// TIA Portal V18 export
// export: Created 2026-06-12T02:00:00Z, ExportSetting WithDefaults, DisplayName Totally Integrated Automation Portal, DisplayVersion V18, DisplayName TIA Portal Openness, DisplayVersion V18
TagTable "HMI_Tags_B3to7"
  AI_B3_Sequence_Count : Real  (PLC tag AI_B3_Sequence_Count, HMI_Connection_1, 1 s)   // 0-100
  AI_B3_Flow_CIP_Center : Real  (PLC tag AI_B3_Flow_CIP_Center, HMI_Connection_1, 1 s)   // 100-200 L/h
  AI_B3_Temp_CIP_Upper : Real  (PLC tag AI_B3_Temp_CIP_Upper, HMI_Connection_1, 1 s)   // 50-80 °C
  AI_B3_Pressure_CIP_1 : Real  (PLC tag AI_B3_Pressure_CIP_1, HMI_Connection_1, 1 s)   // 7.0-8.0 bar
  AI_B3_Temp_Chaff_1 : Real  (PLC tag AI_B3_Temp_Chaff_1, HMI_Connection_1, 1 s)   // 50-80 °C
  AI_B3_Flow_CIP_Feed : Real  (PLC tag AI_B3_Flow_CIP_Feed, HMI_Connection_1, 1 s)   // 100-200 L/h
  AI_B3_Temp_Steam_1 : Real  (PLC tag AI_B3_Temp_Steam_1, HMI_Connection_1, 1 s)   // 50-80 °C
  AI_B3_Flow_UCWW_1 : Real  (PLC tag AI_B3_Flow_UCWW_1, HMI_Connection_1, 1 s)   // 100-200 L/h
  AI_B3_RPM_Screw_Conv : Real  (PLC tag AI_B3_RPM_Screw_Conv, HMI_Connection_1, 1 s)   // 800-1200 RPM
  AI_B3_Temp_Condensate_1 : Real  (PLC tag AI_B3_Temp_Condensate_1, HMI_Connection_1, 1 s)   // 50-80 °C
  AI_B3_Pressure_Screw_1 : Real  (PLC tag AI_B3_Pressure_Screw_1, HMI_Connection_1, 1 s)   // 7.0-8.0 bar
  AI_B3_Flow_CWW_Out : Real  (PLC tag AI_B3_Flow_CWW_Out, HMI_Connection_1, 1 s)   // 100-200 L/h
  AI_B3_Pressure_CWW_1 : Real  (PLC tag AI_B3_Pressure_CWW_1, HMI_Connection_1, 1 s)   // 7.0-8.0 bar
  AI_B3_Temp_Decanter2 : Real  (PLC tag AI_B3_Temp_Decanter2, HMI_Connection_1, 1 s)   // 50-80 °C
  AI_B3_RPM_Rotary2 : Real  (PLC tag AI_B3_RPM_Rotary2, HMI_Connection_1, 1 s)   // 800-1200 RPM
  AI_B3_RPM_Rotary1 : Real  (PLC tag AI_B3_RPM_Rotary1, HMI_Connection_1, 1 s)   // 800-1200 RPM
  AI_B3_Temp_GroundSilo : Real  (PLC tag AI_B3_Temp_GroundSilo, HMI_Connection_1, 1 s)   // 50-80 °C
  AI_B3_Flow_GroundSilo : Real  (PLC tag AI_B3_Flow_GroundSilo, HMI_Connection_1, 1 s)   // 100-200 L/h
  AI_B3_Pressure_Mid_1 : Real  (PLC tag AI_B3_Pressure_Mid_1, HMI_Connection_1, 1 s)   // 7.0-8.0 bar
  AI_B3_Flow_Condensate : Real  (PLC tag AI_B3_Flow_Condensate, HMI_Connection_1, 1 s)   // 100-200 L/h
  AI_B3_Flow_Sump_Out : Real  (PLC tag AI_B3_Flow_Sump_Out, HMI_Connection_1, 1 s)   // 100-200 L/h
  AI_B3_Level_Sump : Real  (PLC tag AI_B3_Level_Sump, HMI_Connection_1, 1 s)   // 30-80 %
  AI_B3_Pressure_Decant1 : Real  (PLC tag AI_B3_Pressure_Decant1, HMI_Connection_1, 1 s)   // 7.0-8.0 bar
  AI_B3_Pressure_Decant2 : Real  (PLC tag AI_B3_Pressure_Decant2, HMI_Connection_1, 1 s)   // 7.0-8.0 bar
  AI_B3_Flow_Decant1 : Real  (PLC tag AI_B3_Flow_Decant1, HMI_Connection_1, 1 s)   // 100-200 L/h
  AI_B3_Temp_Decant1 : Real  (PLC tag AI_B3_Temp_Decant1, HMI_Connection_1, 1 s)   // 50-80 °C
  AI_B3_Temp_FBB_Boiler : Real  (PLC tag AI_B3_Temp_FBB_Boiler, HMI_Connection_1, 1 s)   // 50-80 °C
  AI_B3_Temp_CWW_Out : Real  (PLC tag AI_B3_Temp_CWW_Out, HMI_Connection_1, 1 s)   // 50-80 °C
  AI_B3_Pressure_SUMP : Real  (PLC tag AI_B3_Pressure_SUMP, HMI_Connection_1, 1 s)   // 7.0-8.0 bar
  AI_B3_Flow_SUMP : Real  (PLC tag AI_B3_Flow_SUMP, HMI_Connection_1, 1 s)   // 100-200 L/h
  AI_B3_Level_CWW : Real  (PLC tag AI_B3_Level_CWW, HMI_Connection_1, 1 s)   // 30-80 %
  AI_B3_Temp_FBB_Out : Real  (PLC tag AI_B3_Temp_FBB_Out, HMI_Connection_1, 1 s)   // 50-80 °C
  AI_B3_Pressure_FBB_Out : Real  (PLC tag AI_B3_Pressure_FBB_Out, HMI_Connection_1, 1 s)   // 7.0-8.0 bar
  AI_B3_Flow_FBB_Out : Real  (PLC tag AI_B3_Flow_FBB_Out, HMI_Connection_1, 1 s)   // 100-200 L/h
  AI_B4_Daq_C : Real  (PLC tag AI_B4_Daq_C, HMI_Connection_1, 1 s)   // 0-100
  AI_B4_TPH_Total : Real  (PLC tag AI_B4_TPH_Total, HMI_Connection_1, 1 s)   // 100-200 T/h
  AI_B4_KG_CM_Main : Real  (PLC tag AI_B4_KG_CM_Main, HMI_Connection_1, 1 s)   // 7.0-8.0 kg/cm2
  AI_B4_DRM_LVL1 : Real  (PLC tag AI_B4_DRM_LVL1, HMI_Connection_1, 1 s)   // 30-80 %
  AI_B4_DRM_LVL2 : Real  (PLC tag AI_B4_DRM_LVL2, HMI_Connection_1, 1 s)   // 30-80 %
  AI_B4_MW_Output : Real  (PLC tag AI_B4_MW_Output, HMI_Connection_1, 1 s)   // 0-50 MW
  AI_B4_KG_CM_2 : Real  (PLC tag AI_B4_KG_CM_2, HMI_Connection_1, 1 s)   // 7.0-8.0 kg/cm2
  AI_B4_Hc_Value : Real  (PLC tag AI_B4_Hc_Value, HMI_Connection_1, 1 s)   // 0-100
  AI_B4_Temp_AirHeater_In1 : Real  (PLC tag AI_B4_Temp_AirHeater_In1, HMI_Connection_1, 1 s)   // 50-80 °C
  AI_B4_Temp_AirHeater_In2 : Real  (PLC tag AI_B4_Temp_AirHeater_In2, HMI_Connection_1, 1 s)   // 50-80 °C
  AI_B4_Temp_AirHeater_In3 : Real  (PLC tag AI_B4_Temp_AirHeater_In3, HMI_Connection_1, 1 s)   // 50-80 °C
  AI_B4_Temp_AirHeater_Out1 : Real  (PLC tag AI_B4_Temp_AirHeater_Out1, HMI_Connection_1, 1 s)   // 50-80 °C
  AI_B4_Temp_AirHeater_Out2 : Real  (PLC tag AI_B4_Temp_AirHeater_Out2, HMI_Connection_1, 1 s)   // 50-80 °C
  AI_B4_Pres_AH_mmWC_1 : Real  (PLC tag AI_B4_Pres_AH_mmWC_1, HMI_Connection_1, 1 s)   // 7.0-8.0 mmWC
  AI_B4_Pres_AH_mmWC_2 : Real  (PLC tag AI_B4_Pres_AH_mmWC_2, HMI_Connection_1, 1 s)   // 7.0-8.0 mmWC
  AI_B4_Pres_AH_Pct_1 : Real  (PLC tag AI_B4_Pres_AH_Pct_1, HMI_Connection_1, 1 s)   // 20-80 %
  AI_B4_Temp_AH_Out3 : Real  (PLC tag AI_B4_Temp_AH_Out3, HMI_Connection_1, 1 s)   // 50-80 °C
  AI_B4_Pres_FDH_mmWC : Real  (PLC tag AI_B4_Pres_FDH_mmWC, HMI_Connection_1, 1 s)   // 7.0-8.0 mmWC
  AI_B4_RPM_PAF1 : Real  (PLC tag AI_B4_RPM_PAF1, HMI_Connection_1, 1 s)   // 800-1200 RPM
  AI_B4_Pct_RPC308_SP : Real  (PLC tag AI_B4_Pct_RPC308_SP, HMI_Connection_1, 1 s)   // 20-80 %
  AI_B4_Pct_RPC308_PV : Real  (PLC tag AI_B4_Pct_RPC308_PV, HMI_Connection_1, 1 s)   // 20-80 %
  AI_B4_Pres_PAF1_mmWC : Real  (PLC tag AI_B4_Pres_PAF1_mmWC, HMI_Connection_1, 1 s)   // 7.0-8.0 mmWC
  AI_B4_Pct_FDF1_SP : Real  (PLC tag AI_B4_Pct_FDF1_SP, HMI_Connection_1, 1 s)   // 20-80 %
  AI_B4_Pct_FDF1_PV : Real  (PLC tag AI_B4_Pct_FDF1_PV, HMI_Connection_1, 1 s)   // 20-80 %
  AI_B4_Pct_FDF1_OUT : Real  (PLC tag AI_B4_Pct_FDF1_OUT, HMI_Connection_1, 1 s)   // 20-80 %
  AI_B4_RPM_FDF1 : Real  (PLC tag AI_B4_RPM_FDF1, HMI_Connection_1, 1 s)   // 800-1200 RPM
  AI_B4_Pct_RPC301_SP : Real  (PLC tag AI_B4_Pct_RPC301_SP, HMI_Connection_1, 1 s)   // 20-80 %
  AI_B4_Pct_RPC301_PV : Real  (PLC tag AI_B4_Pct_RPC301_PV, HMI_Connection_1, 1 s)   // 20-80 %
  AI_B4_Pct_RPC301_OUT : Real  (PLC tag AI_B4_Pct_RPC301_OUT, HMI_Connection_1, 1 s)   // 20-80 %
  AI_B4_mA_ESP1 : Real  (PLC tag AI_B4_mA_ESP1, HMI_Connection_1, 1 s)   // 50-200 mA
  AI_B4_mA_ESP2 : Real  (PLC tag AI_B4_mA_ESP2, HMI_Connection_1, 1 s)   // 50-200 mA
  AI_B4_mA_ESP3 : Real  (PLC tag AI_B4_mA_ESP3, HMI_Connection_1, 1 s)   // 50-200 mA
  AI_B4_mA_ESP4 : Real  (PLC tag AI_B4_mA_ESP4, HMI_Connection_1, 1 s)   // 50-200 mA
  AI_B4_V_ESP1 : Real  (PLC tag AI_B4_V_ESP1, HMI_Connection_1, 1 s)   // 0-400 V
  AI_B4_V_ESP2 : Real  (PLC tag AI_B4_V_ESP2, HMI_Connection_1, 1 s)   // 0-400 V
  AI_B4_V_ESP3 : Real  (PLC tag AI_B4_V_ESP3, HMI_Connection_1, 1 s)   // 0-400 V
  AI_B4_V_ESP4 : Real  (PLC tag AI_B4_V_ESP4, HMI_Connection_1, 1 s)   // 0-400 V
  AI_B4_Pct_RPC305_SP : Real  (PLC tag AI_B4_Pct_RPC305_SP, HMI_Connection_1, 1 s)   // 20-80 %
  AI_B4_Pct_RPC305_PV : Real  (PLC tag AI_B4_Pct_RPC305_PV, HMI_Connection_1, 1 s)   // 20-80 %
  AI_B4_RPM_IDF1 : Real  (PLC tag AI_B4_RPM_IDF1, HMI_Connection_1, 1 s)   // 800-1200 RPM
  AI_B4_Pct_RPC305_VFD : Real  (PLC tag AI_B4_Pct_RPC305_VFD, HMI_Connection_1, 1 s)   // 20-80 %
  AI_B4_Pct_FDF2_SP : Real  (PLC tag AI_B4_Pct_FDF2_SP, HMI_Connection_1, 1 s)   // 20-80 %
  AI_B4_Pct_FDF2_PV : Real  (PLC tag AI_B4_Pct_FDF2_PV, HMI_Connection_1, 1 s)   // 20-80 %
  AI_B4_Pct_FDF2_OUT : Real  (PLC tag AI_B4_Pct_FDF2_OUT, HMI_Connection_1, 1 s)   // 20-80 %
  AI_B4_RPM_FDF2 : Real  (PLC tag AI_B4_RPM_FDF2, HMI_Connection_1, 1 s)   // 800-1200 RPM
  AI_B4_Pct_RPC306_SP : Real  (PLC tag AI_B4_Pct_RPC306_SP, HMI_Connection_1, 1 s)   // 20-80 %
  AI_B4_Pct_RPC306_PV : Real  (PLC tag AI_B4_Pct_RPC306_PV, HMI_Connection_1, 1 s)   // 20-80 %
  AI_B4_Pct_RPC306_OUT : Real  (PLC tag AI_B4_Pct_RPC306_OUT, HMI_Connection_1, 1 s)   // 20-80 %
  AI_B4_RPM_IDF2 : Real  (PLC tag AI_B4_RPM_IDF2, HMI_Connection_1, 1 s)   // 800-1200 RPM
  AI_B4_Pct_RPC306_VFD : Real  (PLC tag AI_B4_Pct_RPC306_VFD, HMI_Connection_1, 1 s)   // 20-80 %
  AI_B4_Pres_FDF_mmWC : Real  (PLC tag AI_B4_Pres_FDF_mmWC, HMI_Connection_1, 1 s)   // 7.0-8.0 mmWC
  AI_B4_TEST1_Value : Real  (PLC tag AI_B4_TEST1_Value, HMI_Connection_1, 1 s)   // 0-100
  AI_B4_Pct_PAF1_SP : Real  (PLC tag AI_B4_Pct_PAF1_SP, HMI_Connection_1, 1 s)   // 20-80 %
  AI_B4_Pct_PAF1_PV : Real  (PLC tag AI_B4_Pct_PAF1_PV, HMI_Connection_1, 1 s)   // 20-80 %
  AI_B4_Pres_PAF2_mmWC : Real  (PLC tag AI_B4_Pres_PAF2_mmWC, HMI_Connection_1, 1 s)   // 7.0-8.0 mmWC
  AI_B4_RPM_PAF2 : Real  (PLC tag AI_B4_RPM_PAF2, HMI_Connection_1, 1 s)   // 800-1200 RPM
  AI_B4_Pct_RPC308b_SP : Real  (PLC tag AI_B4_Pct_RPC308b_SP, HMI_Connection_1, 1 s)   // 20-80 %
  AI_B4_Pct_RPC308b_PV : Real  (PLC tag AI_B4_Pct_RPC308b_PV, HMI_Connection_1, 1 s)   // 20-80 %
  AI_B4_Pct_DAM303B_SP : Real  (PLC tag AI_B4_Pct_DAM303B_SP, HMI_Connection_1, 1 s)   // 20-80 %
  AI_B4_Pct_DAM304B_SP : Real  (PLC tag AI_B4_Pct_DAM304B_SP, HMI_Connection_1, 1 s)   // 20-80 %
  AI_B5_CA_Fan_Motor_DE_Temp : Real  (PLC tag AI_B5_CA_Fan_Motor_DE_Temp, HMI_Connection_1, 1 s)   // 50-80 °C
  AI_B5_CA_Fan_Motor_NDE_Temp : Real  (PLC tag AI_B5_CA_Fan_Motor_NDE_Temp, HMI_Connection_1, 1 s)   // 50-80 °C
  AI_B5_CA_Fan_DE_Temp : Real  (PLC tag AI_B5_CA_Fan_DE_Temp, HMI_Connection_1, 1 s)   // 50-80 °C
  AI_B5_CA_Fan_NDE_Temp : Real  (PLC tag AI_B5_CA_Fan_NDE_Temp, HMI_Connection_1, 1 s)   // 50-80 °C
  AI_B5_CA_Fan_DE_Vib : Real  (PLC tag AI_B5_CA_Fan_DE_Vib, HMI_Connection_1, 1 s)   // 0-10 mm/s
  AI_B5_CA_Fan_NDE_Vib : Real  (PLC tag AI_B5_CA_Fan_NDE_Vib, HMI_Connection_1, 1 s)   // 0-10 mm/s
  AI_B5_SP_700FN03 : Real  (PLC tag AI_B5_SP_700FN03, HMI_Connection_1, 1 s)   // 100-200 L/h
  AI_B5_SP_700HES01 : Real  (PLC tag AI_B5_SP_700HES01, HMI_Connection_1, 1 s)   // 100-200 L/h
  AI_B5_SP_700DA4 : Real  (PLC tag AI_B5_SP_700DA4, HMI_Connection_1, 1 s)   // 20-30 Hz
  AI_B5_SP_700DA6 : Real  (PLC tag AI_B5_SP_700DA6, HMI_Connection_1, 1 s)   // 20-30 Hz
  AI_B5_SP_700DA7 : Real  (PLC tag AI_B5_SP_700DA7, HMI_Connection_1, 1 s)   // 20-30 Hz
  AI_B5_SP_700FN2_DA1 : Real  (PLC tag AI_B5_SP_700FN2_DA1, HMI_Connection_1, 1 s)   // 20-30 Hz
  AI_B5_Sep_Motor_Top_Temp : Real  (PLC tag AI_B5_Sep_Motor_Top_Temp, HMI_Connection_1, 1 s)   // 50-80 °C
  AI_B5_Sep_Bottom_Bear_Temp : Real  (PLC tag AI_B5_Sep_Bottom_Bear_Temp, HMI_Connection_1, 1 s)   // 50-80 °C
  AI_B5_Trend_Val_1 : Real  (PLC tag AI_B5_Trend_Val_1, HMI_Connection_1, 1 s)   // 0-100 %
  AI_B5_Trend_Val_2 : Real  (PLC tag AI_B5_Trend_Val_2, HMI_Connection_1, 1 s)   // 0-100 %
  AI_B5_Trend_Val_3 : Real  (PLC tag AI_B5_Trend_Val_3, HMI_Connection_1, 1 s)   // 0-100 %
  AI_B5_700FN03_RPM : Real  (PLC tag AI_B5_700FN03_RPM, HMI_Connection_1, 1 s)   // 800-1200 RPM
  AI_B5_700HES01_Flow : Real  (PLC tag AI_B5_700HES01_Flow, HMI_Connection_1, 1 s)   // 100-200 L/h
  AI_B5_700FN10_Speed : Real  (PLC tag AI_B5_700FN10_Speed, HMI_Connection_1, 1 s)   // 20-30 Hz
  AI_B5_700CM01_Current : Real  (PLC tag AI_B5_700CM01_Current, HMI_Connection_1, 1 s)   // 50-200 A
  AI_B5_Lub_Stop_Time : Real  (PLC tag AI_B5_Lub_Stop_Time, HMI_Connection_1, 1 s)   // 0-300 Sec
  AI_B5_Main_Drive_ReHealth : Real  (PLC tag AI_B5_Main_Drive_ReHealth, HMI_Connection_1, 1 s)   // 0-300 Sec
  AI_B5_CM_LRS_IN : Real  (PLC tag AI_B5_CM_LRS_IN, HMI_Connection_1, 1 s)   // 50-80 °C
  AI_B5_CM_LRS_OUT : Real  (PLC tag AI_B5_CM_LRS_OUT, HMI_Connection_1, 1 s)   // 50-80 °C
  AI_B5_CM_Mill_Oil_Temp : Real  (PLC tag AI_B5_CM_Mill_Oil_Temp, HMI_Connection_1, 1 s)   // 50-80 °C
  AI_B5_CM_OilTrun_BER_Temp : Real  (PLC tag AI_B5_CM_OilTrun_BER_Temp, HMI_Connection_1, 1 s)   // 50-80 °C
  AI_B5_CM_OilTrun_BER2_Temp : Real  (PLC tag AI_B5_CM_OilTrun_BER2_Temp, HMI_Connection_1, 1 s)   // 50-80 °C
  AI_B5_CM_OilPinion_BER_Temp : Real  (PLC tag AI_B5_CM_OilPinion_BER_Temp, HMI_Connection_1, 1 s)   // 50-80 °C
  AI_B5_CM_GB_IL_Shaft_BER : Real  (PLC tag AI_B5_CM_GB_IL_Shaft_BER, HMI_Connection_1, 1 s)   // 50-80 °C
  AI_B5_CM_Running_Hours : Real  (PLC tag AI_B5_CM_Running_Hours, HMI_Connection_1, 1 s)   // 0-8760 Hr
  AI_B5_CM_PS1_1_KG : Real  (PLC tag AI_B5_CM_PS1_1_KG, HMI_Connection_1, 1 s)   // 7-8 bar
  AI_B5_CM_PS1_2_KG : Real  (PLC tag AI_B5_CM_PS1_2_KG, HMI_Connection_1, 1 s)   // 7-8 bar
  AI_B5_NIBS_Value : Real  (PLC tag AI_B5_NIBS_Value, HMI_Connection_1, 1 s)   // 50-200 A
  AI_B5_800DC1_Temp : Real  (PLC tag AI_B5_800DC1_Temp, HMI_Connection_1, 1 s)   // 50-80 °C
  AI_B5_800DC2_Temp : Real  (PLC tag AI_B5_800DC2_Temp, HMI_Connection_1, 1 s)   // 50-80 °C
  AI_B5_800FN1_Speed : Real  (PLC tag AI_B5_800FN1_Speed, HMI_Connection_1, 1 s)   // 20-30 Hz
  AI_B5_800FN2_Speed : Real  (PLC tag AI_B5_800FN2_Speed, HMI_Connection_1, 1 s)   // 20-30 Hz
  AI_B5_800YF1_Flow : Real  (PLC tag AI_B5_800YF1_Flow, HMI_Connection_1, 1 s)   // 100-200 L/h
  AI_B5_800YF2_Flow : Real  (PLC tag AI_B5_800YF2_Flow, HMI_Connection_1, 1 s)   // 100-200 L/h
  AI_B5_Silo1_Level_Bar1 : Real  (PLC tag AI_B5_Silo1_Level_Bar1, HMI_Connection_1, 1 s)   // 0-100 %
  AI_B5_Silo1_Level_Bar2 : Real  (PLC tag AI_B5_Silo1_Level_Bar2, HMI_Connection_1, 1 s)   // 0-100 %
  AI_B5_Silo2_Level_Bar1 : Real  (PLC tag AI_B5_Silo2_Level_Bar1, HMI_Connection_1, 1 s)   // 0-100 %
  AI_B5_Silo2_Level_Bar2 : Real  (PLC tag AI_B5_Silo2_Level_Bar2, HMI_Connection_1, 1 s)   // 0-100 %
  AI_B5_700FN01_Speed : Real  (PLC tag AI_B5_700FN01_Speed, HMI_Connection_1, 1 s)   // 20-30 Hz
  AI_B5_700FN02_Speed : Real  (PLC tag AI_B5_700FN02_Speed, HMI_Connection_1, 1 s)   // 20-30 Hz
  AI_B5_700AS07_Speed : Real  (PLC tag AI_B5_700AS07_Speed, HMI_Connection_1, 1 s)   // 20-30 Hz
  AI_B5_700AS08_Flow : Real  (PLC tag AI_B5_700AS08_Flow, HMI_Connection_1, 1 s)   // 100-200 L/h
  AI_B5_700FN09_Speed : Real  (PLC tag AI_B5_700FN09_Speed, HMI_Connection_1, 1 s)   // 20-30 Hz
  AI_B5_700SFM01_Speed : Real  (PLC tag AI_B5_700SFM01_Speed, HMI_Connection_1, 1 s)   // 20-30 Hz
  AI_B5_700DA1_Flow : Real  (PLC tag AI_B5_700DA1_Flow, HMI_Connection_1, 1 s)   // 100-200 L/h
  AI_B5_700DA4_Flow : Real  (PLC tag AI_B5_700DA4_Flow, HMI_Connection_1, 1 s)   // 100-200 L/h
  AI_B5_700DA6_Temp : Real  (PLC tag AI_B5_700DA6_Temp, HMI_Connection_1, 1 s)   // 50-80 °C
  AI_B5_700DA7_Temp : Real  (PLC tag AI_B5_700DA7_Temp, HMI_Connection_1, 1 s)   // 50-80 °C
  AI_B5_700BL1_Load : Real  (PLC tag AI_B5_700BL1_Load, HMI_Connection_1, 1 s)   // 50-200 A
  AI_B5_700BL2_Load : Real  (PLC tag AI_B5_700BL2_Load, HMI_Connection_1, 1 s)   // 50-200 A
  AI_B5_700AS9_Flow : Real  (PLC tag AI_B5_700AS9_Flow, HMI_Connection_1, 1 s)   // 100-200 L/h
  AI_B5_700FN13_Speed : Real  (PLC tag AI_B5_700FN13_Speed, HMI_Connection_1, 1 s)   // 20-30 Hz
  AI_B6_TICR211_Temp : Real  (PLC tag AI_B6_TICR211_Temp, HMI_Connection_1, 1 s)   // 50-80 °C
  AI_B6_TICR210_Temp : Real  (PLC tag AI_B6_TICR210_Temp, HMI_Connection_1, 1 s)   // 50-80 °C
  AI_B6_TICR201_Tank_Temp : Real  (PLC tag AI_B6_TICR201_Tank_Temp, HMI_Connection_1, 1 s)   // 50-80 °C
  AI_B6_PT201_Pressure : Real  (PLC tag AI_B6_PT201_Pressure, HMI_Connection_1, 1 s)   // 7.0-8.0 bar
  AI_B6_Ph201_pH : Real  (PLC tag AI_B6_Ph201_pH, HMI_Connection_1, 1 s)   // 6.0-8.0 pH
  AI_B6_ORP201_ORP : Real  (PLC tag AI_B6_ORP201_ORP, HMI_Connection_1, 1 s)   // 20-80 %
  AI_B6_DPL101_Level : Real  (PLC tag AI_B6_DPL101_Level, HMI_Connection_1, 1 s)   // 100-500 L
  AI_B6_TICR214_Temp : Real  (PLC tag AI_B6_TICR214_Temp, HMI_Connection_1, 1 s)   // 50-80 °C
  AI_B6_TICR204_Temp : Real  (PLC tag AI_B6_TICR204_Temp, HMI_Connection_1, 1 s)   // 50-80 °C
  AI_B6_TICR205_Temp : Real  (PLC tag AI_B6_TICR205_Temp, HMI_Connection_1, 1 s)   // 50-80 °C
  AI_B6_TICR206_Temp : Real  (PLC tag AI_B6_TICR206_Temp, HMI_Connection_1, 1 s)   // 50-80 °C
  AI_B6_FHC203_Flow : Real  (PLC tag AI_B6_FHC203_Flow, HMI_Connection_1, 1 s)   // 100-200 L/h
  AI_B6_BPC201_Pressure : Real  (PLC tag AI_B6_BPC201_Pressure, HMI_Connection_1, 1 s)   // 7.0-8.0 bar
  AI_B7_K03_PT02_Pressure : Real  (PLC tag AI_B7_K03_PT02_Pressure, HMI_Connection_1, 1 s)   // 7-8 bar
  AI_B7_K03_TT04_Temp : Real  (PLC tag AI_B7_K03_TT04_Temp, HMI_Connection_1, 1 s)   // 50-80 °C
  AI_B7_K03_TT05_Temp : Real  (PLC tag AI_B7_K03_TT05_Temp, HMI_Connection_1, 1 s)   // 50-80 °C
  AI_B7_K03_TT06_Temp : Real  (PLC tag AI_B7_K03_TT06_Temp, HMI_Connection_1, 1 s)   // 50-80 °C
  AI_B7_K03_TT07_Temp : Real  (PLC tag AI_B7_K03_TT07_Temp, HMI_Connection_1, 1 s)   // 50-80 °C
  AI_B7_K03_PT07_Pressure : Real  (PLC tag AI_B7_K03_PT07_Pressure, HMI_Connection_1, 1 s)   // 7-8 bar
  AI_B7_K03_FT03_Flow : Real  (PLC tag AI_B7_K03_FT03_Flow, HMI_Connection_1, 1 s)   // 100-200 L/h
  AI_B7_K03_Density_1 : Real  (PLC tag AI_B7_K03_Density_1, HMI_Connection_1, 1 s)   // 800-1000 kg/m3
  AI_B7_K03_LT01_Level : Real  (PLC tag AI_B7_K03_LT01_Level, HMI_Connection_1, 1 s)   // 20-80 cm
  AI_B7_K03_LT02_Level : Real  (PLC tag AI_B7_K03_LT02_Level, HMI_Connection_1, 1 s)   // 20-80 cm
  AI_B7_K03_TT01_Temp : Real  (PLC tag AI_B7_K03_TT01_Temp, HMI_Connection_1, 1 s)   // 50-80 °C
  AI_B7_K03_TT02_Temp : Real  (PLC tag AI_B7_K03_TT02_Temp, HMI_Connection_1, 1 s)   // 50-80 °C
  AI_B7_Reboiler_PV : Real  (PLC tag AI_B7_Reboiler_PV, HMI_Connection_1, 1 s)   // 100-200 L/h
  AI_B7_Reboiler_SP : Real  (PLC tag AI_B7_Reboiler_SP, HMI_Connection_1, 1 s)   // 100-200 L/h
  AI_B7_Reboiler_CV : Real  (PLC tag AI_B7_Reboiler_CV, HMI_Connection_1, 1 s)   // 20-80 %
  AI_B7_HE03_Primary_Temp : Real  (PLC tag AI_B7_HE03_Primary_Temp, HMI_Connection_1, 1 s)   // 50-80 °C
  AI_B7_HE03_Secondary_Temp : Real  (PLC tag AI_B7_HE03_Secondary_Temp, HMI_Connection_1, 1 s)   // 50-80 °C
  AI_B7_K03_L08_Level : Real  (PLC tag AI_B7_K03_L08_Level, HMI_Connection_1, 1 s)   // 20-80 cm
  AI_B7_K03_L06_Level : Real  (PLC tag AI_B7_K03_L06_Level, HMI_Connection_1, 1 s)   // 20-80 cm
  AI_B7_K03_L05_Level : Real  (PLC tag AI_B7_K03_L05_Level, HMI_Connection_1, 1 s)   // 20-80 cm
  AI_B7_K03_L07_Level : Real  (PLC tag AI_B7_K03_L07_Level, HMI_Connection_1, 1 s)   // 20-80 cm
  AI_B7_K03_L04_Level : Real  (PLC tag AI_B7_K03_L04_Level, HMI_Connection_1, 1 s)   // 20-80 cm
  AI_B7_K03_L03_Level : Real  (PLC tag AI_B7_K03_L03_Level, HMI_Connection_1, 1 s)   // 20-80 cm
  AI_B7_V03A_Density : Real  (PLC tag AI_B7_V03A_Density, HMI_Connection_1, 1 s)   // 800-1000 kg/m3
  AI_B7_Kettle_Flow_SP : Real  (PLC tag AI_B7_Kettle_Flow_SP, HMI_Connection_1, 1 s)   // 100-200 kg/h
  AI_B7_Keboiler_Flow_SP : Real  (PLC tag AI_B7_Keboiler_Flow_SP, HMI_Connection_1, 1 s)   // 100-200 kg/h
  AI_B7_Reflux_Time_SP : Real  (PLC tag AI_B7_Reflux_Time_SP, HMI_Connection_1, 1 s)   // 0-60 Min
  AI_B7_Time_Remain : Real  (PLC tag AI_B7_Time_Remain, HMI_Connection_1, 1 s)   // 0-60 Min
  AI_B7_RD_Level_SP : Real  (PLC tag AI_B7_RD_Level_SP, HMI_Connection_1, 1 s)   // 20-80 cm
  AI_B7_Reflux_Flow_SP : Real  (PLC tag AI_B7_Reflux_Flow_SP, HMI_Connection_1, 1 s)   // 100-200 L/h
  AI_B7_Collection_SP : Real  (PLC tag AI_B7_Collection_SP, HMI_Connection_1, 1 s)   // 100-200 L/h
  AI_B7_Total_Flowrate : Real  (PLC tag AI_B7_Total_Flowrate, HMI_Connection_1, 1 s)   // 100-200 L/h
  AI_B7_ML_Qty_SP : Real  (PLC tag AI_B7_ML_Qty_SP, HMI_Connection_1, 1 s)   // 0-600 L
  AI_B7_ML_Qty_Total : Real  (PLC tag AI_B7_ML_Qty_Total, HMI_Connection_1, 1 s)   // 0-600 L
  AI_B7_Material_Code : Real  (PLC tag AI_B7_Material_Code, HMI_Connection_1, 1 s)   // 0-99
  AI_B7_Stage_Number : Real  (PLC tag AI_B7_Stage_Number, HMI_Connection_1, 1 s)   // 0-20
  AI_B7_Batch_Number : Real  (PLC tag AI_B7_Batch_Number, HMI_Connection_1, 1 s)   // 0-9999
  AI_B7_Current_User_ID : Real  (PLC tag AI_B7_Current_User_ID, HMI_Connection_1, 1 s)   // 0-999
  AI_B7_K_05_L_704_HI : Real  (PLC tag AI_B7_K_05_L_704_HI, HMI_Connection_1, 1 s)   // 20-80 cm
  AI_B7_Density_SP : Real  (PLC tag AI_B7_Density_SP, HMI_Connection_1, 1 s)   // 800-1000 kg/m3
  AI_B7_CTS_Flow_1 : Real  (PLC tag AI_B7_CTS_Flow_1, HMI_Connection_1, 1 s)   // 100-200 kg/h
  AI_B7_CTS_Flow_2 : Real  (PLC tag AI_B7_CTS_Flow_2, HMI_Connection_1, 1 s)   // 100-200 kg/h
  AI_B7_Steam_PT01_Temp : Real  (PLC tag AI_B7_Steam_PT01_Temp, HMI_Connection_1, 1 s)   // 50-80 °C
  AI_B7_Steam_PT02_Temp : Real  (PLC tag AI_B7_Steam_PT02_Temp, HMI_Connection_1, 1 s)   // 50-80 °C
  AI_B7_CWS_TT01_Temp : Real  (PLC tag AI_B7_CWS_TT01_Temp, HMI_Connection_1, 1 s)   // 50-80 °C
  AI_B7_CWS_TT02_Temp : Real  (PLC tag AI_B7_CWS_TT02_Temp, HMI_Connection_1, 1 s)   // 50-80 °C
  AI_B7_CWS_TT03_Temp : Real  (PLC tag AI_B7_CWS_TT03_Temp, HMI_Connection_1, 1 s)   // 50-80 °C
  AI_B7_CWAR_TT01_Temp : Real  (PLC tag AI_B7_CWAR_TT01_Temp, HMI_Connection_1, 1 s)   // 50-80 °C
  AI_B7_CWAR_TT02_Temp : Real  (PLC tag AI_B7_CWAR_TT02_Temp, HMI_Connection_1, 1 s)   // 50-80 °C
  AI_B7_CWAR_TT03_Temp : Real  (PLC tag AI_B7_CWAR_TT03_Temp, HMI_Connection_1, 1 s)   // 50-80 °C
  AI_B7_CWAR_TT04_Temp : Real  (PLC tag AI_B7_CWAR_TT04_Temp, HMI_Connection_1, 1 s)   // 50-80 °C
  AI_B7_K03_CV01_PV : Real  (PLC tag AI_B7_K03_CV01_PV, HMI_Connection_1, 1 s)   // 20-80 %
  AI_B7_K03_CV01_SP : Real  (PLC tag AI_B7_K03_CV01_SP, HMI_Connection_1, 1 s)   // 20-80 %
  AI_B7_K03_CV01_CV : Real  (PLC tag AI_B7_K03_CV01_CV, HMI_Connection_1, 1 s)   // 20-80 %
  AI_B7_Steam_CV01_PV : Real  (PLC tag AI_B7_Steam_CV01_PV, HMI_Connection_1, 1 s)   // 20-80 %
  AI_B7_Steam_CV01_SP : Real  (PLC tag AI_B7_Steam_CV01_SP, HMI_Connection_1, 1 s)   // 20-80 %
  AI_B7_Steam_CV01_CV : Real  (PLC tag AI_B7_Steam_CV01_CV, HMI_Connection_1, 1 s)   // 20-80 %
  AI_B7_K03_Jacket_PV : Real  (PLC tag AI_B7_K03_Jacket_PV, HMI_Connection_1, 1 s)   // 50-80 °C
  AI_B7_K03_Jacket_SP : Real  (PLC tag AI_B7_K03_Jacket_SP, HMI_Connection_1, 1 s)   // 50-80 °C
  AI_B7_K03_Jacket_CV : Real  (PLC tag AI_B7_K03_Jacket_CV, HMI_Connection_1, 1 s)   // 20-80 %
  AI_B7_CHWR_TT01_Temp : Real  (PLC tag AI_B7_CHWR_TT01_Temp, HMI_Connection_1, 1 s)   // 50-80 °C
  AI_B7_CHWR_TT02_Temp : Real  (PLC tag AI_B7_CHWR_TT02_Temp, HMI_Connection_1, 1 s)   // 50-80 °C
  AI_B7_CHWS_TT01_Temp : Real  (PLC tag AI_B7_CHWS_TT01_Temp, HMI_Connection_1, 1 s)   // 50-80 °C
  AI_B7_CHWS_TT02_Temp : Real  (PLC tag AI_B7_CHWS_TT02_Temp, HMI_Connection_1, 1 s)   // 50-80 °C
  AI_B7_K03_TT03_Temp : Real  (PLC tag AI_B7_K03_TT03_Temp, HMI_Connection_1, 1 s)   // 50-80 °C
